PROGRAM P_ParameterComm
VAR
	fbMC_Power: MC_Power;
	fbMC_WriteParameter: MC_WriteParameter;
	bWrite: BOOL;
	fbMC_MoveAbsolute: MC_MoveAbsolute;
	fb_MC_MoveAbsolute: MC_MoveAbsolute;
END_VAR


//This function calls the ReadStatus of the axis.	
kidAxis.ReadStatus();


fbMC_Power(
	Axis:= kidAxis, 
	Enable:= GVL_Modes.bDrive_Enable, 
	Enable_Positive:= , 
	Enable_Negative:= , 
	Override:= GVL_Modes.lrDrive_Override, 
	BufferMode:= , 
	Options:= , 
	Status=> , 
	Busy=> , 
	Active=> , 
	Error=> , 
	ErrorID=> );
	



fbMC_WriteParameter(
	Axis:= kidaxis, 
	Execute:= bWrite, 
	ParameterNumber:= AxisEnPositionLagMonitoring, 
	Value:= 1, 
	Done=> , 
	Busy=> , 
	Error=> , 
	ErrorID=> );
	
fbMC_MoveAbsolute.Position := GVL_Index.Target_Down;
	
	
fbMC_MoveAbsolute(
	Axis:= kidAxis, 
	Execute:= bStart_Motion, 
	Position:= , 
	Velocity:= 360, 
	Acceleration:= , 
	Deceleration:= , 
	Jerk:= , 
	BufferMode:= , 
	Options:= , 
	Done=> , 
	Busy=> , 
	Active=> , 
	CommandAborted=> , 
	Error=> , 
	ErrorID=> );

ACTION A_MC_MoveAbsolute:




fb_MC_MoveAbsolute(
	Axis:= kidAxis, 
	Execute:= bStart_Motion, 
	Position:= 0, 
	Velocity:= , 
	Acceleration:= , 
	Deceleration:= , 
	Jerk:= , 
	BufferMode:= , 
	Options:= , 
	Done=> , 
	Busy=> , 
	Active=> , 
	CommandAborted=> , 
	Error=> , 
	ErrorID=> );
END_ACTION

END_PROGRAM

(* stored: Version 1.1.0.1, ProductVersion 3.1.4022.3
   POU P_ParameterComm: Id {8375a1a9-74c4-4479-9932-6deb80094c2a}, SpecialFunc None
   Action A_MC_MoveAbsolute: Id {617cf1b6-5be2-46ff-bdaa-f96c512dd327} *)
